{attribute 'GeneratedUsingTerminal: ATH2050-5501-0022'}
{attribute addProperty BoxType "ATH2050-5501-0022"}
{attribute addProperty Id "FB_InputsAT %I*FB_Inputs_391456510FB_OutputsAT %Q*FB_Outputs_DAFD38E02WcStateAT %I*WcState_9091E0EB2InfoDataAT %I*InfoData_A7436BC610"}
{attribute addProperty CRC "1858116023"}
{attribute addProperty Size "14"}
TYPE ATH2050_6EC099B7 EXTENDS EtcSlaveTerminalBase_947E5A46 :
STRUCT
	{attribute addProperty Name "FB_Inputs"}
	FB_Inputs : FB_Inputs_39145651;
	{attribute addProperty Name "FB_Outputs"}
	FB_Outputs : FB_Outputs_DAFD38E0;
	{attribute addProperty Name "WcState"}
	WcState : WcState_9091E0EB;
	{attribute addProperty Name "InfoData"}
	InfoData : InfoData_A7436BC6;
END_STRUCT
END_TYPE

(* stored: Version 1.2.0.0, ProductVersion 3.1.4024.9
   DUT ATH2050_6EC099B7: Id {4fc2e475-d65e-49eb-b67e-b6abaa824b8a} *)
